                               //save last requested ROI coordinates
                               //-----------------------------------
                               #center_x_old        :=  #set_center_x;
                               #center_y_old        :=  #set_center_y;
                               #outer_radius_old    :=  #set_outer_radius;
                               #inner_radius_old    :=  #set_inner_radius;
                               #start_angle_old     :=  #set_start_angle;
                               #stop_angle_old      :=  #set_stop_angle;
                            END_IF;
                       END_IF;

                   //stero camera mode
                   //-----------------
                   ELSE
                       //ROI stereo camera 1
                       //-------------------
                       #set_ctr_x_scam_1    :=  "CM_INSELECT"(auto    :=  "APC".AUTOMATIC,              // area in x-dimension
                                                           track   :=  TRUE,
                                                           ac      :=  ROUND("AC".SET_ROI_CTR_X_SCAM),
                                                           kya     :=  "KYA".SET_ROI_CTR_X_SCAM);

                       #set_ctr_y_scam_1    :=  "CM_INSELECT"(auto    :=  "APC".AUTOMATIC,              //area in y-dimension
                                                           track   :=  TRUE,
                                                           ac      :=  ROUND("AC".SET_ROI_CTR_Y_SCAM),
                                                           kya     :=  "KYA".SET_ROI_CTR_Y_SCAM);

                       #set_width_scam_1    :=  "CM_INSELECT"(auto    :=  "APC".AUTOMATIC,              //sensor width
                                                           track   :=  TRUE,
                                                           ac      :=  ROUND("AC".SET_SEN_HGT),      //sensor rotated 90? height and width exchanged
                                                           kya     :=  "KYA".SET_ROI_HGT_SCAM);

                       #set_height_scam_1   :=  "CM_INSELECT"(auto    :=  "APC".AUTOMATIC,              //sensor height
                                                           track   :=  TRUE,
                                                           ac      :=  ROUND("AC".SET_SEN_WDH),      //sensor rotated 90? height and width exchanged
                                                           kya     :=  "KYA".SET_ROI_WDH_SCAM);

                       //check if ROI coordinate change is requested
                       //-------------------------------------------
                       IF NOT #O_NEW_ROI_CRD  THEN
                           //sensor position change stereo camera 1
                           //--------------------------------------
                           IF  (#set_ctr_x_scam_1 <> #set_ctr_x_scam_1_old)  OR
                               (#set_ctr_y_scam_1 <> #set_ctr_y_scam_1_old)  OR
                               (#set_width_scam_1 <> #set_width_scam_1_old)  OR
                               (#set_height_scam_1 <> #set_height_scam_1_old)    THEN 

                               #new_roi_crd :=  true;

                               //convert parameter values in string variables
                               //-------------------------------------------- 
                               #ctr_x_scam1     :=  DINT_TO_STRING (IN:= REAL_TO_DINT(#set_ctr_x_scam_1 * 100));
                               #ctr_y_scam1     :=  DINT_TO_STRING (IN:= REAL_TO_DINT(#set_ctr_y_scam_1 * 100));    
                               #width_scam1     :=  DINT_TO_STRING (IN:= REAL_TO_DINT(#set_width_scam_1 * 100));
                               #height_scam1    :=  DINT_TO_STRING (IN:= REAL_TO_DINT(#set_height_scam_1 * 100));    

                           END_IF;
                           //evaluate new ROI coordinate command string
                           //------------------------------------------
                           IF #new_roi_crd THEN

                               //delete ROI coordinate string
                               //----------------------------   
                               #roi_crd_strg := DELETE(IN:= #roi_crd_strg, L:= 60, P:= 0);

                               //built new ROI coordinate string
                               //-------------------------------     
                               #roi_crd_strg    := CONCAT(IN1:= 'rke1_cc=' , IN2:= #ctr_x_scam1);

                               #roi_crd_strg    := CONCAT(IN1:= #roi_crd_strg, IN2:= #delimiter);

                               #roi_crd_strg    := CONCAT(IN1:= #roi_crd_strg, IN2:= #ctr_y_scam1);

                               #roi_crd_strg    := CONCAT(IN1:= #roi_crd_strg, IN2:= #delimiter);

                               #roi_crd_strg    := CONCAT(IN1:= #roi_crd_strg, IN2:= #width_scam1);

                               #roi_crd_strg    := CONCAT(IN1:= #roi_crd_strg, IN2:= #delimiter);

                               #roi_crd_strg    := CONCAT(IN1:= #roi_crd_strg, IN2:= #height_scam1);

                               #O_ROI_CRD_STRG  :=  #roi_crd_strg;    //write new ROI coordinate string
                               #O_NEW_ROI_CRD   :=  true;

                               //save last requested ROI coordinates
                               //-----------------------------------
                               #set_ctr_x_scam_1_old    :=  #set_ctr_x_scam_1;
                               #set_ctr_y_scam_1_old    :=  #set_ctr_y_scam_1;
                               #set_width_scam_1_old    :=  #set_width_scam_1;
                               #set_height_scam_1_old   :=  #set_height_scam_1;
                           END_IF;
                       END_IF;

                       //ROI stereo camera 2
                       //-------------------
                       #set_ctr_x_scam_2    :=  #set_ctr_x_scam_1 + "PAR_SUB".CTR_X_SCAM_2_ADJ;
                       #set_ctr_y_scam_2    :=  #set_ctr_y_scam_1 + "PAR_SUB".CTR_Y_SCAM_2_ADJ;
                       #set_width_scam_2    :=  #set_width_scam_1;
                       #set_height_scam_2   :=  #set_height_scam_1;

                       //check if ROI coordinate change is requested
                       //-------------------------------------------
                       IF NOT #O_NEW_ROI_CRD  THEN
                           //sensor position change stereo camera 2
                           //--------------------------------------
                           IF  (#set_ctr_x_scam_2 <> #set_ctr_x_scam_2_old)  OR
                               (#set_ctr_y_scam_2 <> #set_ctr_y_scam_2_old)  OR
                               (#set_width_scam_2 <> #set_width_scam_2_old)  OR
                               (#set_height_scam_2 <> #set_height_scam_2_old)    THEN 

                               #new_roi_crd :=  true;

                               //convert parameter values in string variables
                               //-------------------------------------------- 
                               #ctr_x_scam2     :=  DINT_TO_STRING (IN:= REAL_TO_DINT(#set_ctr_x_scam_2 * 100));
                               #ctr_y_scam2     :=  DINT_TO_STRING (IN:= REAL_TO_DINT(#set_ctr_y_scam_2 * 100));    
                               #width_scam2     :=  DINT_TO_STRING (IN:= REAL_TO_DINT(#set_width_scam_2 * 100));
                               #height_scam2    :=  DINT_TO_STRING (IN:= REAL_TO_DINT(#set_height_scam_2 * 100));    

                           END_IF;
                           //evaluate new ROI coordinate command string
                           //------------------------------------------
                           IF #new_roi_crd THEN

                               //delete ROI coordinate string
                               //----------------------------   
                               #roi_crd_strg := DELETE(IN:= #roi_crd_strg, L:= 60, P:= 0);

                               //built new ROI coordinate string
                               //-------------------------------     
                               #roi_crd_strg    := CONCAT(IN1:= 'rke2_cc=' , IN2:= #ctr_x_scam2);

                               #roi_crd_strg    := CONCAT(IN1:= #roi_crd_strg, IN2:= #delimiter);

                               #roi_crd_strg    := CONCAT(IN1:= #roi_crd_strg, IN2:= #ctr_y_scam2);

                               #roi_crd_strg    := CONCAT(IN1:= #roi_crd_strg, IN2:= #delimiter);

                               #roi_crd_strg    := CONCAT(IN1:= #roi_crd_strg, IN2:= #width_scam2);

                               #roi_crd_strg    := CONCAT(IN1:= #roi_crd_strg, IN2:= #delimiter);

                               #roi_crd_strg    := CONCAT(IN1:= #roi_crd_strg, IN2:= #height_scam2);

                               #O_ROI_CRD_STRG  :=  #roi_crd_strg;    //write new ROI coordinate string
                               #O_NEW_ROI_CRD   :=  true;

                               //save last requested ROI coordinates
                               //-----------------------------------
                               #set_ctr_x_scam_2_old    :=  #set_ctr_x_scam_2;
                               #set_ctr_y_scam_2_old    :=  #set_ctr_y_scam_2;
                               #set_width_scam_2_old    :=  #set_width_scam_2;
                               #set_height_scam_2_old   :=  #set_height_scam_2;
                           END_IF;
                       END_IF;
                   END_IF;        

               //rectangle ROI is selected
               //-------------------------
               ELSIF "LT".CAM_PRD_1_SEL THEN
                   #set_center_x    :=  "CM_INSELECT"(auto    :=  "APC".AUTOMATIC,              // area in x-dimension
                                                   track   :=  TRUE,
                                                   ac      :=  ROUND("AC".SET_SEN_CTR_X),
                                                   kya     :=  "KYA".SET_SEN_CTR_X_P1);

                   #set_center_y    :=  "CM_INSELECT"(auto    :=  "APC".AUTOMATIC,              //area in y-dimension
                                                   track   :=  TRUE,
                                                   ac      :=  ROUND("AC".SET_SEN_CTR_Y),
                                                   kya     :=  "KYA".SET_SEN_CTR_Y_P1);

                   #set_width       :=  "CM_INSELECT"(auto    :=  "APC".AUTOMATIC,              //sensor width
                                                   track   :=  TRUE,
                                                   ac      :=  ROUND("AC".SET_SEN_WDH),
                                                   kya     :=  "KYA".SET_SEN_WDH_P1);


                   #set_height       :=  "CM_INSELECT"(auto   :=  "APC".AUTOMATIC,              //sensor height
                                                   track   :=  TRUE,
                                                   ac      :=  ROUND("AC".SET_SEN_HGT),
                                                   kya     :=  "KYA".SET_SEN_HGT_P1);


                   //check if ROI coordinate change is requested
                   //-------------------------------------------
                   IF NOT #O_NEW_ROI_CRD  THEN
                       //melting detection
                       //-----------------
                       IF  (#set_center_x <> #center_x_old)  OR
                           (#set_center_y <> #center_y_old)  OR
                           (#set_width <> #width_old)        OR
                           (#set_height <> #height_old)      THEN 

                           #new_roi_crd :=  true;

                           //convert parameter values in string variables
                           //-------------------------------------------- 
                           #center_x    :=  DINT_TO_STRING (IN:= REAL_TO_DINT(#set_center_x * 100));
                           #center_y    :=  DINT_TO_STRING (IN:= REAL_TO_DINT(#set_center_y * 100));    
                           #width       :=  DINT_TO_STRING (IN:= REAL_TO_DINT(#set_width * 100));
                           #height      :=  DINT_TO_STRING (IN:= REAL_TO_DINT(#set_height * 100));    

                       END_IF;
                   END_IF;

                   //evaluate new ROI coordinate command string
                   //------------------------------------------
                   IF #new_roi_crd THEN

                       //delete ROI coordinate string
                       //----------------------------   
                       #roi_crd_strg := DELETE(IN:= #roi_crd_strg, L:= 60, P:= 0);

                       //built new ROI coordinate string
                       //-------------------------------     
                       #roi_crd_strg    := CONCAT(IN1:= 'rec_crd=' , IN2:= #center_x);

                       #roi_crd_strg    := CONCAT(IN1:= #roi_crd_strg, IN2:= #delimiter);

                       #roi_crd_strg    := CONCAT(IN1:= #roi_crd_strg, IN2:= #center_y);

                       #roi_crd_strg    := CONCAT(IN1:= #roi_crd_strg, IN2:= #delimiter);

                       #roi_crd_strg    := CONCAT(IN1:= #roi_crd_strg, IN2:= #width);

                       #roi_crd_strg    := CONCAT(IN1:= #roi_crd_strg, IN2:= #delimiter);

                       #roi_crd_strg    := CONCAT(IN1:= #roi_crd_strg, IN2:= #height);

                       #O_ROI_CRD_STRG  :=  #roi_crd_strg;    //write new ROI coordinate string
                       #O_NEW_ROI_CRD   :=  true;

                       //save last requested ROI coordinates
                       //-----------------------------------
                       #center_x_old    :=  #set_center_x;
                       #center_y_old    :=  #set_center_y;
                       #width_old       :=  #set_width;
                       #height_old      :=  #set_height;

                   END_IF;
               END_IF; 
           END_IF;

           //reset flag new ROI coordinates
           //------------------------------
           #new_roi_crd :=  false;

           //melt vibration measurement - acitve in all measurement methods
           //--------------------------------------------------------------
           //read settings of melt vibration sensor from recipe or manual input 
           //------------------------------------------------------------------
           #set_mlt_vib_center_x    :=  "KYA".SET_SEN_MLT_VIB_CTR_X;          //area in y-dimension

           #set_mlt_vib_center_y    :=  "KYA".SET_SEN_MLT_VIB_CTR_Y;          //area in y-dimension

           #set_mlt_vib_width       :=  "KYA".SET_SEN_MLT_VIB_WDH;            //senor width

           //check if ROI coordinate change is requested
           //-------------------------------------------
           IF NOT #O_NEW_ROI_CRD  THEN
               //melt vibration measurement
               //--------------------------
               IF (#set_mlt_vib_center_x <> #mlt_vib_center_x_old)  OR
                  (#set_mlt_vib_center_y <> #mlt_vib_center_y_old)  OR
                  (#set_mlt_vib_width <> #mlt_vib_width_old)        THEN 

                   #new_mlt_vib_roi_crd :=  true;

                   //convert parameter values in string variables
                   //-------------------------------------------- 
                   #mlt_vib_center_x    :=  DINT_TO_STRING (IN:= REAL_TO_DINT(#set_mlt_vib_center_x * 100));
                   #mlt_vib_center_y    :=  DINT_TO_STRING (IN:= REAL_TO_DINT(#set_mlt_vib_center_y * 100));    
                   #mlt_vib_width       :=  DINT_TO_STRING (IN:= REAL_TO_DINT(#set_mlt_vib_width * 100));

               END_IF; 
           END_IF;       

           //evaluate new melt vibration ROI coordinate command string
           //---------------------------------------------------------
           IF #new_mlt_vib_roi_crd THEN

               //delete ROI coordinate string
               //----------------------------   
               #roi_crd_strg := DELETE(IN:= #roi_crd_strg, L:= 60, P:= 0);

               //built new ROI coordinate string
               //-------------------------------     
               #roi_crd_strg    := CONCAT(IN1:= 'vib_crd=' , IN2:= #mlt_vib_center_x);

               #roi_crd_strg    := CONCAT(IN1:= #roi_crd_strg, IN2:= #delimiter);

               #roi_crd_strg    := CONCAT(IN1:= #roi_crd_strg, IN2:= #mlt_vib_center_y);

               #roi_crd_strg    := CONCAT(IN1:= #roi_crd_strg, IN2:= #delimiter);

               #roi_crd_strg    := CONCAT(IN1:= #roi_crd_strg, IN2:= #mlt_vib_width);

               #O_ROI_CRD_STRG  :=  #roi_crd_strg;    //write new ROI coordinate string
               #O_NEW_ROI_CRD   :=  true;

               //save last requested ROI coordinates
               //-----------------------------------
               #mlt_vib_center_x_old    :=  #set_mlt_vib_center_x;
               #mlt_vib_center_y_old    :=  #set_mlt_vib_center_y;
               #mlt_vib_width_old       :=  #set_mlt_vib_width;

               //reset flag new melt vibration ROI coordinates
               //---------------------------------------------
               #new_mlt_vib_roi_crd :=  false;

           END_IF;     

           //evaluate recipe threshold setpoint
           //----------------------------------
           #ac_set_sen_thr  :=  ROUND("AC".SET_SEN_THR * 10.0);   //shift decimal place one digit to the right and round

           #ac_set_sen_thr  :=  #ac_set_sen_thr / 10.0;          //shift decimal place one digit to the left 

           //evaluate recipe threshold setpoint for camera 2
           //----------------------------------
           #ac_set_sen_thr_2  :=  ROUND("AC".SET_CAM_2_THR * 10.0);   //shift decimal place one digit to the right and round

           #ac_set_sen_thr_2  :=  #ac_set_sen_thr_2 / 10.0;          //shift decimal place one digit to the left 

           //evaluate threshold setpoint mode related
           //----------------------------------------
           IF "LT".CAM_MLT   THEN
               //read sensor threshold
               //---------------------
               #set_thr :=  "CM_INSELECT"(auto    :=  "APC".AUTOMATIC,              
                                       track   :=  TRUE,
                                       ac      :=  #ac_set_sen_thr,             //use rounded value
                                       kya     :=  "KYA".SET_SEN_THR_P4);

               //set command identifier
               //----------------------
               #thr_cmd         :=  'mlt_thr=';

           ELSIF "LT".CAM_DIP   THEN
               //read sensor threshold
               //---------------------
               #set_thr :=  "CM_INSELECT"(auto    :=  "APC".AUTOMATIC,              
                                       track   :=  TRUE,
                                       ac      :=  #ac_set_sen_thr,             //use rounded value
                                       kya     :=  "KYA".SET_SEN_THR_P3);

               //set command identifier
               //----------------------
               #thr_cmd         :=  'dip_thr=';

           ELSIF "LT".CAM_DIA   THEN
               //read threshold of seqmented circle ROI
               //--------------------------------------           
               IF "LT".CAM_PRD_2_SEL THEN 
                   //threshold
                   //---------
                   #set_thr :=  "CM_INSELECT"(auto    :=  "APC".AUTOMATIC,              
                                           track   :=  TRUE,
                                           ac      :=  #ac_set_sen_thr,             //use rounded value
                                           kya     :=  "KYA".SET_SEN_THR_P2);

                   //set circle sensor command identifier
                   //------------------------------------
                   #thr_cmd         :=  'dia_thr=';

                   //stereo camera installed
                   //-----------------------
                   IF (("CNF".ACT_DVC_CNF AND 2#0000_0000_0000_1000_0000_0000_0000_0000) = 2#0000_0000_0000_1000_0000_0000_0000_0000) THEN  
                       //shoulder phase
                       //--------------
                       IF ("APC".STATUS = "APC".SHOULDER) THEN
                           //threshold - used for a second camera only in shoulder phase
                           //-----------------------------------------------------------
                           #set_thr_2 :=  "CM_INSELECT"(auto    :=  "APC".AUTOMATIC,              
                                                     track   :=  TRUE,
                                                     ac      :=  #ac_set_sen_thr_2,             //use rounded value
                                                     kya     :=  "KYA".SET_CAM_2_THR);

                           //set circle sensor command identifier
                           //------------------------------------
                           #thr_cmd_2        :=  'diathr2=';
                       //other phases
                       //------------
                       ELSE
                           "KYA".SET_CAM_2_THR   := #set_thr; //track KYA value of second threshold with first threshold      
                       END_IF;
                   END_IF;    
               //read threshold of rectangle ROI
               //-------------------------------
               ELSIF "LT".CAM_PRD_1_SEL  THEN 
                   #set_thr :=  "CM_INSELECT"(auto    :=  "APC".AUTOMATIC,              
                                           track   :=  TRUE,
                                           ac      :=  #ac_set_sen_thr,             //use rounded value
                                           kya     :=  "KYA".SET_SEN_THR_P1);

                   //set circle sensor command identifier
                   //------------------------------------
                   #thr_cmd         :=  'rec_thr=';

               END_IF;
           END_IF;

           //read melt vibration sensor threshold
           //------------------------------------
           #set_mlt_vib_thr :=  "KYA".SET_SEN_MLT_VIB_THR;

           //check if ROI threshold change is requested
           //------------------------------------------
           IF NOT #O_NEW_ROI_THR THEN
               //melting, dipping or diameter measurement
               //----------------------------------------
               IF (#set_thr <> #thr_old) THEN 
                   #new_thr_req :=  true;

                   //convert parameter values in string variables
                   //-------------------------------------------- 
                   #thr :=  INT_TO_STRING (IN:= REAL_TO_INT(#set_thr * 100));      //circle sensor, dip line or junk detection

               //melt vibration measurement
               //--------------------------
               ELSIF (#set_mlt_vib_thr <> #mlt_vib_thr_old) THEN
                   #new_mlt_vib_thr_req :=  true;

                   //convert melt vibration threshold parameter value in string variable
                   //------------------------------------------------------------------- 
                   #mlt_vib_thr :=  INT_TO_STRING (IN:= REAL_TO_INT(#set_mlt_vib_thr * 100));

               END_IF; 
           END_IF;

           //check if ROI threshold change is requested for camera 2
           //------------------------------------------
           IF NOT #O_NEW_ROI_THR_2 THEN
               //melting, dipping or diameter measurement
               //----------------------------------------

               IF (#set_thr_2 <> #thr_old_2) THEN 
                   #new_thr_req_2 :=  true;

                   //convert parameter values in string variables
                   //-------------------------------------------- 
                   #thr_2 :=  INT_TO_STRING (IN:= REAL_TO_INT(#set_thr_2 * 100));      //circle sensor, dip line or junk detection

               END_IF;        
           END_IF;

           //evaluate new ROI threshold command string
           //-----------------------------------------
           IF #new_thr_req THEN                         //melting, dipping or diameter measurement

               //delete command string
               //---------------------   
               #roi_thr_strg := DELETE(IN:= #roi_thr_strg, L:= 20, P:= 0);

               //built new command string
               //------------------------     
               #roi_thr_strg    := CONCAT(IN1:= #thr_cmd, IN2:= #thr);

               #O_ROI_THR_STRG  :=  #roi_thr_strg;    //write new ROI threshold string
               #O_NEW_ROI_THR   :=  true;

               //save last requested sensor threshold parameter
               //----------------------------------------------
               #thr_old :=  #set_thr;

               //reset new sensor shape flag
               //--------------------------- 
               #new_thr_req :=  false;


           ELSIF #new_mlt_vib_thr_req THEN              //melt vibration measurement

               //delete command string
               //---------------------   
               #roi_thr_strg := DELETE(IN:= #roi_thr_strg, L:= 20, P:= 0);

               //built new command string
               //------------------------     
               #roi_thr_strg    := CONCAT(IN1:= 'vib_thr=', IN2:= #mlt_vib_thr);

               #O_ROI_THR_STRG  :=  #roi_thr_strg;    //write new ROI threshold string
               #O_NEW_ROI_THR   :=  true;

               //save last requested sensor threshold parameter
               //----------------------------------------------
               #mlt_vib_thr_old :=  #set_mlt_vib_thr;

               //reset new sensor shape flag
               //--------------------------- 
               #new_mlt_vib_thr_req :=  false;


           END_IF;

           //evaluate new ROI threshold command string for camnera 2
           //-----------------------------------------

           IF #new_thr_req_2 THEN                         //melting, dipping or diameter measurement

               //delete command string
               //---------------------   
               #roi_thr_strg_2 := DELETE(IN:= #roi_thr_strg_2, L:= 20, P:= 0);

               //built new command string
               //------------------------     
               #roi_thr_strg_2    := CONCAT(IN1:= #thr_cmd_2, IN2:= #thr_2);

               #O_ROI_THR_STRG_2  :=  #roi_thr_strg_2;    //write new ROI threshold string
               #O_NEW_ROI_THR_2   :=  true;

               //save last requested sensor threshold parameter
               //----------------------------------------------
               #thr_old_2 :=  #set_thr_2;

               //reset new sensor shape flag
               //--------------------------- 
               #new_thr_req_2 :=  false;
           END_IF;


       END_IF;
END_FUNCTION_BLOCK

FUNCTION_BLOCK "CHAR_TO_DINT"   // FB104, SCL
{ S7_Optimized_Access := 'FALSE' }
VERSION : 0.0
// --------------------------------------------------------------------------------
//     program     :    CHAR_TO_DINT
//     description :    convert characters to double integer      
//     name        :    G. Eibelsh鋟ser
//     date        :    11.05.2010
// 
//     revision    :
//     name        :
//     date        :    
//                     (c)PVA Tepla AG
//     --------------------------------------------------------------------------------
   VAR_INPUT
      I_AMT_OF_BYTES : Int;
   END_VAR
   VAR_OUTPUT
      O_CAM_VALUE : Array[0..19] of DInt;   // increased for stereo camera test
   END_VAR
   VAR
      i : Int;
      k : Int;
      digit : Int;
      number : DInt;
   END_VAR
BEGIN

       //init temporary function variables
       //---------------------------------
       #digit      := 0;                                   
       #number     := 0;
       #k          := 0;

       FOR #i:= 4 TO (#I_AMT_OF_BYTES) DO        //exclude first four characters in data DB                             
           //last character detected - abort calculation and function
           //--------------------------------------------------------
           IF "BM_CAM_EVAL_DB".Data[#i] = BYTE_TO_CHAR(B#16#D) THEN        //exit conversion when carriage return appears in telegram
               #O_CAM_VALUE[#k] := #number;
               EXIT;
           ELSE
               //delimter detected - abort calculation of value
               //----------------------------------------------
               IF ("BM_CAM_EVAL_DB".Data[#i] = ';')THEN             
                   #O_CAM_VALUE[#k]  := #number;
                   #k               := #k + 1;                               //increase value counter
                   #number          := 0;
                   #digit           := 0;
               //calculate double integer from characters byte wise
               //--------------------------------------------------
               ELSE
                   #digit := CHAR_TO_INT("BM_CAM_EVAL_DB".Data[#i])-48;   // convert ASCII character in integer value
                   #number   := #number * 10 + #digit;                       
               END_IF;
           END_IF;
       END_FOR;
END_FUNCTION_BLOCK

FUNCTION_BLOCK "BM_MOB_FDR_MAIN"   // FB105, SCL
{ S7_Optimized_Access := 'FALSE' }
VERSION : 0.0
// --------------------------------------------------------------------------------
//     program     :   BM_MOB_FDR_MAIN
//     description :   main control of mobile feeder
//     name        :   G. Eibelsh鋟ser
//     date        :   26.10.2011
//   
//     revision    :
//     name        :
//     date        :    
//                     (c)PVATePla AG
//     --------------------------------------------------------------------------------
   VAR
      i : Int;
   END_VAR
   VAR_TEMP
      dbl_srv_mode : Bool;
   END_VAR
BEGIN

       //ReadStatus from feeder
       //-------------------------------------------------------------------------
       "DV".CB_FLT_AC230V_FDR  := DWORD_TO_DINT("P_BM_FDR_STAT":P AND 2#0000_0000_0000_0001)<>0;
       "DV".CB_FLT_DC24V_FDR   := DWORD_TO_DINT("P_BM_FDR_STAT":P AND 2#0000_0000_0000_0010)<>0;
       "DV".FDR_CH_HOME_POS    := DWORD_TO_DINT("P_BM_FDR_STAT":P AND 2#0000_0000_0000_0100)<>0;
       "DV".FDR_CH_FDG_POS     := DWORD_TO_DINT("P_BM_FDR_STAT":P AND 2#0000_0000_0000_1000)<>0;
       "DV".FDR_TUBE_HOME_POS  := DWORD_TO_DINT("P_BM_FDR_STAT":P AND 2#0000_0000_0001_0000)<>0;
       "DV".FDR_TUBE_FCH_POS   := DWORD_TO_DINT("P_BM_FDR_STAT":P AND 2#0000_0000_0010_0000)<>0;
       "DV".FDR_TUBE_FDG_POS   := DWORD_TO_DINT("P_BM_FDR_STAT":P AND 2#0000_0000_0100_0000)<>0;
       "DV".FDR_IN_POS         := DWORD_TO_DINT("P_BM_FDR_STAT":P AND 2#0000_0000_1000_0000)<>0;

       //                      := DV.FDR_VIB_ENB  

       //reset feeder undocking done flag when feeder is electrically disconnected
       //-------------------------------------------------------------------------
       IF NOT "DV".MOB_FDR_CON    THEN 
           "LT".MOB_FDR_UDCK_DONE    :=  FALSE; 
           "DV".MOB_FDR_PB_TRM       :=  FALSE;               
           #i                       :=  0;

       //reset mobile feeder connection flag before electrical disconnection
       //-------------------------------------------------------------------
       ELSIF "LT".MOB_FDR_UDCK_DONE THEN
           //IF BYTE_TO_INT(PEB256)<>0 THEN
           //    DV.MOB_FDR_PB_TRM   :=  FALSE;
           //END_IF;                  
           #i   :=  0;

       //set mobile feeder connection flag
       //---------------------------------
       ELSIF "DV".MOB_FDR_CON THEN                  //electrical connection done
           IF (#i > 50) THEN 
               "DV".MOB_FDR_PB_TRM   :=  TRUE;       //termination flag 5s delayed               
           ELSE
               IF "SysTick100ms" THEN 
                   #i   :=  #i + 1;
               END_IF;
           END_IF;
       END_IF;

       //electrical connection of mobile feeder done
       //-------------------------------------------
       "LT".MOB_FDR_EL_CON_DONE  :=  "DV".MOB_FDR_PB_TRM;

       //disable service mode when sequences are active
       //----------------------------------------------
       #dbl_srv_mode    :=  "APC".AUTOMATIC OR "LT".MOB_FDR_DCK_ATV OR "LT".MOB_FDR_UDCK_ATV OR "LT".MOB_FDR_MVE_IN_SEQ_ON OR "LT".MOB_FDR_MVE_OUT_SEQ_ON;

       //activate/deactivate service mode of mobile feeder
       //-------------------------------------------------
       IF #dbl_srv_mode THEN 
           "LT".MOB_FDR_SRV_ON :=    FALSE;
       ELSE
           "LT".MOB_FDR_SRV_ON := ("KYD".MOB_FDR_SRV_ON OR "LT".MOB_FDR_SRV_ON) AND NOT "KYD".MOB_FDR_SRV_OFF;
       END_IF;

       //call mobile feeder modules
       //--------------------------
       IF "DV".MOB_FDR_CALL THEN 
           //service function activated
           //--------------------------
           IF "LT".MOB_FDR_SRV_ON THEN
               //call mobile feeder service function
               //-----------------------------------
               "BM_MOB_FDR_SRV"();
           ELSE            
               //call mobile feeder drive sequence function block
               //------------------------------------------------
               "BM_MOB_FDR_DRV_SEQ_DB"();

           END_IF; 

           //set circuit breaker alarm messages of mobile feeder
           //---------------------------------------------------
           "FLT".MOB_FDR_CB_AC_230V  := "DV".CB_FLT_AC230V_FDR;

           "FLT".MOB_FDR_CB_DC_24V   := "DV".CB_FLT_DC24V_FDR;                

           //write status variables
           //----------------------
           "LT".MOB_FDR_CH_HOME_POS  :=  "DV".FDR_CH_HOME_POS;
           "LT".MOB_FDR_TUBE_HOME_POS:=  "DV".FDR_TUBE_HOME_POS;
           "LT".MOB_FDR_TUBE_FCH_POS :=  "DV".FDR_TUBE_FCH_POS;
           "LT".MOB_FDR_CH_FDG_POS   :=  "DV".FDR_CH_FDG_POS;
           "LT".MOB_FDR_TUBE_FDG_POS :=  "DV".FDR_TUBE_FDG_POS;
           "LT".FDR_LS_TUBE_OUT      :=  "DV".FDR_TUBE_HOME_POS;    //used for tube symbol in EKZ Explorer

           //write display values of mobile feeder
           //-------------------------------------
           "DIS".MOB_FDR_ACT_TUBE_TMP    :=  0.0;
           "DIS".MOB_FDR_ACT_TUBE_POS    :=  "P_BM_FDR_ACT_TUBE_POS":P;
           "DIS".ACT_LEAKR_FDR           :=  "AV".MOB_FDR_LKR;    //AV.AVG_FDG_RTE; 
           "DIS".ACT_PRS_DROP_FDR        :=  "AV".ACT_PRS_DROP_FDR;
           "DIS".MOB_FDR_ACT_CRG_LVL     :=  "P_BM_FDR_ACT_CRG_LVL":P;

       ELSE
           //reset circuit breaker alarm messages of mobile feeder
           //---------------------------------------------------
           "FLT".MOB_FDR_CB_AC_230V      :=  FALSE;
           "FLT".MOB_FDR_CB_DC_24V       :=  FALSE;

           "FLT".MOB_FDR_INIT_KL_3312    :=  FALSE;  
           "FLT".MOB_FDR_TC_TUBE         :=  FALSE;  
           "FLT".MOB_FDR_INIT_KL2552     :=  FALSE; 
           "FLT".MOB_FDR_MOV_IN_SEQ_ABR  :=  FALSE; 
           "FLT".MOB_FDR_MOV_OUT_SEQ_ABR :=  FALSE; 
           "FLT".MOB_FDR_DCK_SEQ_ABR     :=  FALSE;
           "FLT".MOB_FDR_UDCK_SEQ_ABR    :=  FALSE;
           "FLT".MOB_FDR_FNC_PRS_HI      :=  FALSE;
           "FLT".MOB_FDR_PRS_HI          :=  FALSE;
           "FLT".FEED_RTE_TOO_HI         :=  FALSE;

           //reset vacuum control flags
           //--------------------------
           "DV".MOB_FDR_P3_ON_REQ        :=  FALSE;
           "DV".MOB_FDR_V3_2_OPN_REQ     :=  FALSE;
           "DV".MOB_FDR_V24_OPN_REQ      :=  FALSE;

           //reset status variables
           //----------------------
           "LT".MOB_FDR_CH_HOME_POS  :=  FALSE;
           "LT".MOB_FDR_TUBE_HOME_POS:=  FALSE;

           "LT".MOB_FDR_TUBE_FCH_POS :=  FALSE;

           "LT".MOB_FDR_CH_FDG_POS   :=  FALSE;
           "LT".MOB_FDR_TUBE_FDG_POS :=  FALSE;

           "LT".MOB_FDR_TUBE_DN      :=  FALSE;
           "LT".MOB_FDR_TUBE_UP      :=  FALSE;
           "LT".MOB_FDR_TUBE_STOP    :=  FALSE;
           "LT".MOB_FDR_CH_SW_R      :=  FALSE;
           "LT".MOB_FDR_CH_SW_L      :=  FALSE;
           "LT".MOB_FDR_CH_SW_STOP   :=  FALSE;

           //reset display values of mobile feeder
           //-------------------------------------
           "DIS".MOB_FDR_ACT_TUBE_POS    :=  0.0;
           "DIS".MOB_FDR_SET_VIB_FRQ     :=  0.0;
           "DIS".MOB_FDR_ACT_CRG_LVL     :=  0.0;
           "DIS".ACT_STD_DEV_FILL_LVL    :=  0.0;

           //call mobile feeder service function
           //-----------------------------------
           IF "LT".MOB_FDR_SRV_ON THEN
               "BM_MOB_FDR_SRV"();
           END_IF;
       END_IF;


       //check if mobile feeder is located on puller flange
       //--------------------------------------------------
       IF "DV".FDR_IN_POS THEN
           IF NOT "LT".MOB_FDR_IN_POS THEN 
               //reset mobile feeder docking and drive sequence variables
               //-------------------------------------------------------- 
               "LT".MOB_FDR_DCK_ATV          :=  FALSE;
               "LT".MOB_FDR_UDCK_ATV         :=  FALSE;
               "LT".MOB_FDR_DCK_DONE         :=  FALSE;
               "LT".MOB_FDR_UDCK_DONE        :=  FALSE;
               "LT".MOB_FDR_MVE_OUT_SEQ_ON   :=  FALSE;
               "LT".MOB_FDR_MVE_IN_SEQ_ON    :=  FALSE;
               "LT".MOB_FDR_MVE_SEQ_ARB      :=  FALSE;        
               "LT".MOB_FDR_TUBE_DN          :=  FALSE;
               "LT".MOB_FDR_TUBE_UP          :=  FALSE;
               "LT".MOB_FDR_TUBE_STOP        :=  FALSE;
               "LT".MOB_FDR_CH_SW_R          :=  FALSE;
               "LT".MOB_FDR_CH_SW_L          :=  FALSE;
               "LT".MOB_FDR_CH_SW_STOP       :=  FALSE;
               "LT".MOB_FDR_VIB_ON           :=  FALSE;
           END_IF;
           "LT".MOB_FDR_IN_POS   :=  TRUE;
       ELSE
           "LT".MOB_FDR_IN_POS   :=  FALSE;
       END_IF;
END_FUNCTION_BLOCK

FUNCTION_BLOCK "BM_MOB_FDR_DCK"   // FB106, SCL
{ S7_Optimized_Access := 'FALSE' }
VERSION : 0.0
// --------------------------------------------------------------------------------
//     program     :   BM_MOB_FDR_DCK
//     description :   docking of mobile feeder to puller
//     name        :   G. Eibelsh鋟ser
//     date        :   26.10.2011
//   
//     revision    :
//     name        :
//     date        :    
//                     (c)PVATePla AG
//     --------------------------------------------------------------------------------
   VAR
      arb_dck_seq : Bool;
      "step" : Int;
      i : Int;
      j : Int;
      prg_cnt : Int;
      mob_fdr_prs_bfe_lt : Real;
   END_VAR
BEGIN

       //set mobile feeder docking request 
       //---------------------------------
       IF          "LT".MOB_FDR_IN_POS                   //mobile feeder is in position
           AND NOT "LT".MOB_FDR_UDCK_ATV                 //undocking sequence is not running
           AND NOT "LT".MOB_FDR_DCK_DONE                 //docking sequence is not done
           AND NOT "LT".MOB_FDR_UDCK_DONE    THEN        //undocking sequence is not done - reseted after disconnection of plug

           IF "KYD".MOB_FDR_DCK_ON  THEN
               "LT".MOB_FDR_DCK_ATV  :=  TRUE;
           END_IF;
       END_IF;

       //abort mobile feeder docking sequence and vent feeder
       //----------------------------------------------------
       IF NOT "LT".MOB_FDR_DCK_DONE  AND NOT "FLT".MOB_FDR_DCK_SEQ_ABR THEN
           IF "LT".MOB_FDR_DCK_ATV AND "KYD".MOB_FDR_ARB_SEQ  THEN
               #arb_dck_seq  :=  true;
           END_IF;
       END_IF;

       //mobile feeder docking sequence
       //------------------------------
       IF "LT".MOB_FDR_DCK_ATV  THEN 

           //set step to abort docking sequence
           //----------------------------------
           IF (#arb_dck_seq AND (#step <> 90)) THEN
               #step    := 90;
           END_IF;

           //sequence steps
           //--------------
           CASE #step OF 

               0 : //initialisation step
                   //-------------------
                   #i                       :=  0;
                   #prg_cnt                 :=  0;
                   "AV".MOB_FDR_LKR          :=  0.0;
                   "AV".ACT_PRS_DROP_FDR     :=  0.0;
                   "FLT".ME_LEAK_TST_FDR     :=  FALSE;
                   "FLT".MOB_FDR_DCK_SEQ_ABR :=  FALSE;
                   "FLT".MOB_FDR_UDCK_SEQ_ABR:=  FALSE;
                   "FLT".MOB_FDR_PMP_TME     :=  FALSE;
                   "DV".MOB_FDR_V11_OPN_REQ  :=  FALSE;
                   "DV".MOB_FDR_V11_CLD_REQ  :=  TRUE;
                   "DV".FDG_MVE_IN_SEQ_DONE  :=  FALSE;
                   #step                    :=  #step + 10;

               10: //switch on vacuum pump P3 and open valve V3.2
                   //--------------------------------------------
                   "DV".MOB_FDR_P3_ON_REQ    :=  TRUE;
                   IF "SysTick1s"    THEN
                       #i := #i + 1;
                   END_IF;

                   IF (#i > 3) THEN                     //wait 
                       "DV".MOB_FDR_V3_2_OPN_REQ :=  TRUE;
                   END_IF;

                   IF ("DV".MOB_FDR_V3_2_OPN_REQ AND "PDO".V3_2) THEN                    //valve V3.2 opened
                       #step    :=  #step + 10;
                       #i       :=  0;
                       #j       :=  0;
                   END_IF;

               20: //pump down of mobile feeder
                   //--------------------------
                   IF (REAL_TO_INT("PAR_MAIN".MOB_FDR_DCK_PRG_CYC) > 0) THEN            //check amount of purge cycles 
                       IF ("AV".ACT_PRS_FDR <= "PAR_MAIN".MOB_FDR_DCK_PRG_PRS) THEN
                           #step    :=  #step + 10;
                       END_IF;
                       // Monitoring pump time
                       IF "SysTick1s" THEN
                          #j := #j+1;
                       END_IF;

                       IF (#j> REAL_TO_INT("PAR_MAIN".MOB_FDR_DCK_ALM_TME1)) THEN
                          "FLT".MOB_FDR_PMP_TME := ("AV".ACT_PRS_FDR > "PAR_MAIN".MOB_FDR_DCK_PRS_TRG1);
                       ELSE                  
                          "FLT".MOB_FDR_PMP_TME := False;
                       END_IF;
                       IF (#j> REAL_TO_INT("PAR_MAIN".MOB_FDR_DCK_ALM_TME2))THEN
                          "FLT".MOB_FDR_PMP_TME := ("AV".ACT_PRS_FDR > "PAR_MAIN".MOB_FDR_DCK_PRS_TRG2);
                       ELSE                  
                          "FLT".MOB_FDR_PMP_TME := False;
                       END_IF;

                   //pump down without purging
                   //-------------------------
                   ELSE
                       #step    :=  #step + 30;      //pump down to final pressure
                   END_IF;

               30: //close feeder vacuum valve V3.2
                   //------------------------------
                   "DV".MOB_FDR_V3_2_OPN_REQ :=  FALSE;
                   "FLT".MOB_FDR_PMP_TME := False;

                   IF "SysTick1s"    THEN
                       #i := #i + 1;
                   END_IF;

                   IF NOT "PDO".V3_2 THEN                    //valve V3.2 closed
                       IF (#i > 3) THEN                     //wait 
                           #step    :=  #step + 10;
                           #prg_cnt :=  #prg_cnt + 1;
                           #i       :=  0;
                       END_IF;
                   END_IF;

               40: //purge feeder
                   //------------       
                   IF (#i >= (REAL_TO_INT("PAR_MAIN".MOB_FDR_DCK_PRG_TME)) OR "DV".APS_FDR_DELAYED) THEN
                       "DV".MOB_FDR_V24_OPN_REQ :=  FALSE;
                   ELSE
                       "DV".MOB_FDR_V24_OPN_REQ :=  TRUE;
                   END_IF;

                   IF "SysTick1s"    THEN
                       #i := #i + 1;
                   END_IF;

                   IF NOT "DV".MOB_FDR_V24_OPN_REQ THEN 
                       IF NOT "PDO".V24 THEN
                           IF (#prg_cnt >= (REAL_TO_INT("PAR_MAIN".MOB_FDR_DCK_PRG_CYC))) THEN  
                               #step    :=  #step + 10;
                               #i       :=  0;
                           ELSE
                               #step    :=  #step - 30;     //repeat pump down and purging
                               #i       :=  0;
                           END_IF;
                       END_IF;     
                   END_IF;
                   #j  := 0;

               50: //pump down to final pressure
                   //---------------------------
                   IF ("AV".ACT_PRS_FDR <= "PAR_MAIN".MOB_FDR_DCK_FIN_PRS) THEN            //final pressure reached
                       IF "SysTick1s" THEN
                           #i := #i+1;
                       END_IF;
                       //wait time before leak test
                       //--------------------------
                       IF (#i >= (REAL_TO_INT("PAR_MAIN".MOB_FDR_DCK_WAIT_TME))) THEN
                           "DV".MOB_FDR_V3_2_OPN_REQ :=  FALSE;
                       END_IF;

                   ELSE
                       "DV".MOB_FDR_V3_2_OPN_REQ :=  TRUE;
                       #i                       :=  0;
                   END_IF;

                   IF NOT ("DV".MOB_FDR_V3_2_OPN_REQ OR "PDO".V3_2) THEN
                       #step    :=  #step + 10;
                       #i       :=  0;
                   END_IF;

                   // Monitoring pump time
                   IF "SysTick1s" THEN
                       #j := #j+1;
                   END_IF;

                   IF (#j> REAL_TO_INT("PAR_MAIN".MOB_FDR_DCK_ALM_TME1)) THEN
                       "FLT".MOB_FDR_PMP_TME := ("AV".ACT_PRS_FDR > "PAR_MAIN".MOB_FDR_DCK_PRS_TRG1);
                   ELSE                  
                       "FLT".MOB_FDR_PMP_TME := False;
                   END_IF;
                   IF (#j> REAL_TO_INT("PAR_MAIN".MOB_FDR_DCK_ALM_TME2))THEN
                       "FLT".MOB_FDR_PMP_TME := ("AV".ACT_PRS_FDR > "PAR_MAIN".MOB_FDR_DCK_PRS_TRG2);
                   ELSE                  
                       "FLT".MOB_FDR_PMP_TME := False;
                   END_IF;


               60: //wait 3 sec after vacuum valve V3.2 is closed and store actual pressure
                   //----------------------------------------------------------------------
                   #mob_fdr_prs_bfe_lt  := "AV".ACT_PRS_FDR; 
                   "FLT".MOB_FDR_PMP_TME := False;

                   IF "SysTick1s"    THEN
                       #i := #i + 1;
                   END_IF;

                   IF (#i > 3) THEN
                       "DV".MOB_FDR_P3_ON_REQ    :=  FALSE;          //switch off pump P3
                       #step                    :=  #step + 10;
                       #i                       :=  0;
                   END_IF;

               70: //leak test -> leakrate = (p2-p1)*V/t
                   //-----------------------------------
                   IF "SysTick1s"    THEN
                       #i := #i + 1;
                   END_IF;

                   //calculate leak rate
                   //-------------------
                   IF (#i > 0) THEN 
                       "AV".MOB_FDR_LKR := ("AV".ACT_PRS_FDR - #mob_fdr_prs_bfe_lt) * "CNF".VOLUME_MOB_FDR / (INT_TO_REAL(#i));
                   END_IF;

                   //keep leak rate on zero if calculation is negative
                   //-------------------------------------------------
                   IF ("AV".MOB_FDR_LKR < 0.0) THEN
                       "AV".MOB_FDR_LKR := 0.0;
                   END_IF;

                   //leak test time over
                   //-------------------
                   IF (#i >= (REAL_TO_INT("PAR_MAIN".MOB_FDR_DCK_LKT_TME))) THEN
                       #step    :=  #step + 10;
                   END_IF;

               80: //set alarm message if leak test failed
                   //-------------------------------------
                   IF ("AV".MOB_FDR_LKR > "PAR_MAIN".MOB_FDR_DCK_MAX_LKR) THEN
                       "FLT".ME_LEAK_TST_FDR :=  TRUE;

                       //repeat leak test
                       //----------------
                       IF "KYD".MOB_FDR_NEW_LKT   THEN
                           #step    :=  #step - 80;      //initialisation step 
                       END_IF;

                       //ignore bad leak rate
                       //--------------------
                       IF "KYD".MOB_FDR_IGN_LEAK_RTE   THEN
                           #step    :=  #step + 30;      //finish sequence
                       END_IF;

                       //abort sequence and vent feeder
                       //------------------------------
                       IF "KYD".MOB_FDR_ARB_SEQ   THEN
                           #step    :=  #step + 10;      //abort sequence
                       END_IF;

                   ELSE
                       #step    :=  #step + 30;          //finish sequence
                   END_IF;

               90: //abort docking sequence and vent feeder
                   //--------------------------------------
                   "DV".MOB_FDR_P3_ON_REQ    :=  FALSE;
                   "DV".MOB_FDR_V3_2_OPN_REQ :=  FALSE;
                   "FLT".MOB_FDR_DCK_SEQ_ABR :=  TRUE;
                   #arb_dck_seq             :=  false;

                   IF "DV".APS_FDR_DELAYED THEN                  //feeder at atmospheric pressure
                       "DV".MOB_FDR_V24_OPN_REQ  :=  FALSE;      //stop venting
                   ELSE 
                       "DV".MOB_FDR_V24_OPN_REQ  :=  TRUE;       //vent feeder
                   END_IF;

                   IF NOT ("DV".MOB_FDR_V24_OPN_REQ OR "PDO".V24) THEN
                       #step    :=  #step + 10;
                   END_IF;

               100://sequence aborted
                   //----------------
                   "LT".MOB_FDR_DCK_DONE :=  FALSE;
                   "LT".MOB_FDR_DCK_ATV  :=  FALSE;
                   "FLT".ME_LEAK_TST_FDR :=  FALSE;
                   #step                :=  0;

               110://finish sequence
                   //---------------
                   "LT".MOB_FDR_DCK_DONE :=  TRUE;
                   "LT".MOB_FDR_DCK_ATV  :=  FALSE;
                   "FLT".ME_LEAK_TST_FDR :=  FALSE;
                   #step                :=  0;

           END_CASE;

       ELSE
           #step    := 0;

       END_IF;
END_FUNCTION_BLOCK

FUNCTION_BLOCK "BM_MOB_FDR_UDCK"   // FB107, SCL
{ S7_Optimized_Access := 'FALSE' }
VERSION : 0.0
// --------------------------------------------------------------------------------
//     program     :   BM_MOB_FDR_UDCK
//     description :   undocking of mobile feeder from puller
//     name        :   G. Eibelsh鋟ser
//     date        :   26.10.2011
//   
//     revision    :
//     name        :
//     date        :    
//                     (c)PVATePla AG
//     --------------------------------------------------------------------------------
   VAR
      arb_udck_seq : Bool;
      fdr_prs_inc_done : Bool;
      "step" : Int;
      i : Int;
      prg_cnt : Int;
      fdr_prs_bfe_prs_drop : Real;
   END_VAR
   VAR CONSTANT
      up_prs_lim : Real := 90.0;
   END_VAR
BEGIN


       //set mobile feeder undocking request 
       //-----------------------------------
       IF      NOT "LT".MOB_FDR_DCK_ATV                                  //feeder docking sequence is not running
           AND NOT "LT".MOB_FDR_UDCK_DONE                                //undocking sequence is not done
           AND     "DV".FDR_TUBE_HOME_POS                             //feeder tube is in home position
           AND     "PDI".LS_V11_CL   THEN                                //valve V11 is closed

           IF "KYD".MOB_FDR_UDCK_ON THEN
               "LT".MOB_FDR_UDCK_ATV  :=  TRUE;
           END_IF;
       END_IF;

       //abort mobile feeder undocking sequence
       //--------------------------------------
       IF NOT "LT".MOB_FDR_UDCK_DONE AND NOT "FLT".MOB_FDR_UDCK_SEQ_ABR THEN
           IF "LT".MOB_FDR_UDCK_ATV AND "KYD".MOB_FDR_ARB_SEQ  THEN
               #arb_udck_seq  :=  true;
           END_IF;
       END_IF;

       //mobile feeder undocking sequence
       //--------------------------------
       IF "LT".MOB_FDR_UDCK_ATV  THEN 

           //set step to abort undocking sequence
           //------------------------------------
           IF #arb_udck_seq THEN
               #step    := 80;      //abort step
           END_IF;

           //sequence steps
           //--------------
           CASE #step OF 

               0 : //initialisation step
                   //-------------------
                   #i                           :=  0;
                   "AV".ACT_PRS_DROP_FDR         :=  0.0;
                   "FLT".ME_PRS_DROP_FDR         :=  FALSE;
                   "FLT".MOB_FDR_FNC_PRS_HI      :=  FALSE;
                   "FLT".MOB_FDR_PRS_HI          :=  FALSE;
                   "FLT".MOB_FDR_DCK_SEQ_ABR     :=  FALSE;
                   "FLT".MOB_FDR_UDCK_SEQ_ABR    :=  FALSE;
                   #fdr_prs_inc_done            :=  false;
                   #step                        :=  #step + 10;

               10: //check if feeder is already at atmospheric pressure
                   //--------------------------------------------------
                   IF "PDI".FDR_APS THEN
                       #step    :=  #step + 60;      //go to step 70 and finish sequence
                   ELSE
                       #step    :=  #step + 10;      //go to next step and check pressure
                   END_IF;

               20: //check if furnace and feeder pressure are in valid range for pressure drop test 
                   //------------------------------------------------------------------------------
                   (*
                   IF ((AV.ACT_PRS_CLF + CNF.MOB_FDR_PRS_INC) >= up_prs_lim) THEN
                       FLT.MOB_FDR_FNC_PRS_HI  :=  TRUE;   
                   ELSIF (AV.ACT_PRS_FDR >= up_prs_lim) THEN
                       FLT.MOB_FDR_PRS_HI  :=  TRUE;   
                   ELSE
                       step    :=  step + 10;      //go to next step and perform sequence
                   END_IF;
                   *)
                   //pressure range test skipped - pressure increase in step30 up to predefined value
                   //--------------------------------------------------------------------------------
                   #step    :=  #step + 10;      //go to next step and perform sequence

               30: //increase feeder pressure
                   //------------------------
                   IF (("AV".ACT_PRS_FDR >= "CNF".MOB_FDR_PRS_INC) OR #fdr_prs_inc_done) THEN
                       "DV".MOB_FDR_V24_OPN_REQ  :=  FALSE;      
                       #fdr_prs_inc_done        :=  true;
                       IF "SysTick1s"    THEN
                           #i := #i + 1;
                       END_IF;

                       IF (#i > 30) THEN                                    //wait 30 seconds
                           #fdr_prs_bfe_prs_drop    :=  "AV".ACT_PRS_FDR;     //store actual feeder pressure
                           #step                    :=  #step + 10;
                           #i                       :=  0;
                       END_IF;
                   ELSE
                       "DV".MOB_FDR_V24_OPN_REQ  :=  TRUE;       //insert gas
                   END_IF;

               40: //V11 pressure drop test
                   //----------------------
                   IF "SysTick1s"    THEN
                       #i := #i + 1;
                   END_IF;

                   //calculate feeder pressure drop
                   //------------------------------
                   "AV".ACT_PRS_DROP_FDR := #fdr_prs_bfe_prs_drop - "AV".ACT_PRS_FDR;

                   //pressure drop time over
                   //-----------------------
                   IF (#i >= (REAL_TO_INT("PAR_MAIN".MOB_FDR_UDCK_LKT_TME))) THEN
                       #step    :=  #step + 10;
                   END_IF;

               50: //set alarm message if pressure drop test failed
                   //----------------------------------------------
                   IF ("AV".ACT_PRS_DROP_FDR > "PAR_MAIN".MOB_FDR_UDCK_MAX_PRS_DRP) THEN
                       "FLT".ME_PRS_DROP_FDR :=  TRUE;       //pressure drop too large - leakage of valve V11

                       //repeat  pressure drop test
                       //----------------
                       IF "KYD".MOB_FDR_NEW_LKT   THEN
                           #step    :=  #step - 50;      //initialisation step 
                       END_IF;

                       //ignore bad leak rate
                       //--------------------
                       IF "KYD".MOB_FDR_IGN_LEAK_RTE   THEN
                           #step    :=  #step + 10;      //finish sequence
                       END_IF;

                       //abort sequence and vent feeder
                       //------------------------------
                       IF "KYD".MOB_FDR_ARB_SEQ   THEN
                           #step    :=  #step + 30;      //abort sequence
                       END_IF;

                   ELSE
                       #step    :=  #step + 10;              //finish sequence
                   END_IF;

               60: //vent feeder
                   //-----------
                   IF "DV".APS_FDR_DELAYED THEN                  //feeder at atmospheric pressure
                       "DV".MOB_FDR_V24_OPN_REQ  :=  FALSE;      //stop venting
                   ELSE 
                       "DV".MOB_FDR_V24_OPN_REQ  :=  TRUE;       //vent feeder
                   END_IF;

                   IF NOT ("DV".MOB_FDR_V24_OPN_REQ OR "PDO".V24)   THEN
                       #step    :=  #step + 10;
                   END_IF;

               70: //finish sequence
                   //---------------
                   "LT".MOB_FDR_UDCK_DONE    :=  TRUE;           //set set feeder undocking done flag
                   "LT".MOB_FDR_DCK_DONE     :=  FALSE;          //reset feeder docking done flag
                   "LT".MOB_FDR_UDCK_ATV     :=  FALSE;
                   "FLT".ME_PRS_DROP_FDR     :=  FALSE;
                   #step                    :=  0;

               80 ://sequence aborted
                   //----------------
                   "FLT".MOB_FDR_UDCK_SEQ_ABR    :=  TRUE;
                   "DV".MOB_FDR_V24_OPN_REQ      :=  FALSE;
                   "LT".MOB_FDR_UDCK_DONE        :=  FALSE;
                   "LT".MOB_FDR_UDCK_ATV         :=  FALSE;
                   #arb_udck_seq                :=  false;
                   #step                        :=  0;

           END_CASE;

       ELSE
           #step    := 0;

       END_IF;
END_FUNCTION_BLOCK

FUNCTION_BLOCK "BM_MOB_FDR_DRV_SEQ"   // FB108, SCL
{ S7_Optimized_Access := 'FALSE' }
VERSION : 0.0
// --------------------------------------------------------------------------------
//     program     :   BM_MOB_FDR_DRV_SEQ
//     description :   drive sequence of mobile feeder
//     name        :   G. Eibelsh鋟ser
//     date        :   31.10.2011
//   
//     revision    :
//     name        :
//     date        :    
//                     (c)PVATePla AG
//     --------------------------------------------------------------------------------
   VAR
      mob_fdr_mve_out_seq_on : Bool;
      fdr_prs_inc_done : Bool;
      i : Int;
      "step" : Int;
      mob_fdr_mve_out_dly : Int;
      cool_dn_stp : Int;
      act_tube_pos_bfe : Real;
   END_VAR
   VAR CONSTANT
      max_prs_hyst : Real := 5.0;   // [mbar]
      prs_inc : Real := 3.0;   // [mbar]
   END_VAR
BEGIN


       //activate feeder tube move sequences
       //-----------------------------------
       IF "LT".MOB_FDR_DCK_DONE THEN
           //trigger sequence abort
           //----------------------
           IF NOT "APC".AUTOMATIC AND ("LT".MOB_FDR_MVE_IN_SEQ_ON XOR "LT".MOB_FDR_MVE_OUT_SEQ_ON) THEN
               IF "KYD".MOB_FDR_MVE_SEQ_ARB OR NOT "PDI".EMO THEN 
                   "LT".MOB_FDR_MVE_SEQ_ARB  :=  TRUE;
               END_IF;
           END_IF;

           IF NOT ("LT".MOB_FDR_MVE_IN_SEQ_ON OR "LT".MOB_FDR_MVE_OUT_SEQ_ON) THEN     
               //automatic mode
               //--------------
               IF "APC".AUTOMATIC THEN
                   //trigger move in sequence
                   //------------------------
                   IF ("DC".MOB_FDR_MVE_IN_SEQ_ON AND NOT "DV".FDG_MVE_IN_SEQ_DONE) THEN
                       "LT".MOB_FDR_MVE_IN_SEQ_ON    :=  TRUE;
                       "LT".MOB_FDR_MVE_SEQ_ARB      :=  FALSE;
                       #step                        :=  0;
                   //trigger move out sequence
                   //------------------------
                   ELSIF ("DC".MOB_FDR_MVE_OUT_SEQ_ON AND NOT "DV".FDG_MVE_OUT_SEQ_DONE AND NOT "LT".MOB_FDR_VIB_ON) THEN
                       "LT".MOB_FDR_MVE_OUT_SEQ_ON   :=  TRUE;
                       "LT".MOB_FDR_MVE_SEQ_ARB      :=  FALSE;
                       #step                        :=  0;
                   END_IF;
               //manual mode
               //-----------
               ELSE
                   //trigger move in sequence
                   //------------------------
                   IF ("KYD".MOB_FDR_MVE_IN_SEQ_ON AND NOT "DV".FDG_MVE_IN_SEQ_DONE) THEN
                       "LT".MOB_FDR_MVE_IN_SEQ_ON    :=  TRUE;
                       "LT".MOB_FDR_MVE_SEQ_ARB      :=  FALSE;
                       #step                        :=  0;
                   //trigger move out sequence
                   //------------------------
                   ELSIF ("KYD".MOB_FDR_MVE_OUT_SEQ_ON AND NOT "DV".FDG_MVE_OUT_SEQ_DONE AND NOT "LT".MOB_FDR_VIB_ON) THEN
                       "LT".MOB_FDR_MVE_OUT_SEQ_ON   :=  TRUE;
                       "LT".MOB_FDR_MVE_SEQ_ARB      :=  FALSE;
                       #step                        :=  0;
                   END_IF;
               END_IF;
           END_IF;
       END_IF;

       //delay tube move out sequence start
       //----------------------------------
       #mob_fdr_mve_out_seq_on  := "SysOndelay"(  DIN     := "LT".MOB_FDR_MVE_OUT_SEQ_ON,   // trigger input
                                               SetTime := 30,                          // setp. time
                                               ActTime := #mob_fdr_mve_out_dly,         // act. time
                                               Tick    := "SysTick100ms");               // timebase (100ms)

       //quartz tube move in furnace sequence
       //------------------------------------
       IF "LT".MOB_FDR_MVE_IN_SEQ_ON THEN

           //abort move in sequence
           //----------------------
           IF "LT".MOB_FDR_MVE_SEQ_ARB THEN
               #step    :=  100;            //abort step
           END_IF;

           //sequence steps
           //-------------- 
           CASE #step OF 

               0 : //initialisation step
                   //-------------------
                   #i                           :=  0;
                   #step                        :=  #step + 10;
                   #fdr_prs_inc_done            :=  false;
                   "DV".FDG_MVE_OUT_SEQ_DONE     :=  FALSE;
                   "FLT".MOB_FDR_MOV_IN_SEQ_ABR  :=  FALSE;          //reset alarm message
                   "FLT".MOB_FDR_MOV_OUT_SEQ_ABR :=  FALSE;          //reset alarm message

               10: //check pressure
                   //--------------
                   IF (("AV".ACT_PRS_FDR <= ("AV".ACT_PRS_FCH + #max_prs_hyst)) OR "PDI".LS_V11_OP) THEN       //feeder pressure above puller pressure
                       #step    :=  #step + 30;      //switch to pressure equalisation step                   
                   ELSE
                       #step    :=  #step + 10;      //switch to next step                    
                   END_IF;

               20: //pump down feeder
                   //----------------
                   IF ("AV".ACT_PRS_FDR <= ("AV".ACT_PRS_FCH )) THEN   
                       "DV".MOB_FDR_V3_2_OPN_REQ :=  FALSE;                      //close valve V3.2
                       #step                    :=  #step + 10;                  //switch to next step
                   ELSE
                       "DV".MOB_FDR_P3_ON_REQ    :=  TRUE;                       //switch on pump
                       "DV".MOB_FDR_V3_2_OPN_REQ :=  TRUE;                       //open valve V3.2
                   END_IF;

               30: //wait 3sec.
                   //----------
                   IF NOT "PDO".V3_2 THEN                            //valve V3.2 closed
                       IF "SysTick1s" THEN
                           #i := #i + 1;                             //increase timer
                       END_IF;
                       IF (#i >= 3) THEN                            //wait 3 sec.
                           #step                    :=  #step + 10;  //switch to next step
                           "DV".MOB_FDR_P3_ON_REQ    :=  FALSE;      //switch off pump
                           #i                       :=  0;
                       END_IF;
                   END_IF;             

               40: //pressure equalisation feeder - puller
                   //-------------------------------------
                   IF (("AV".ACT_PRS_FDR >= ("AV".ACT_PRS_FCH + #prs_inc)) OR #fdr_prs_inc_done OR "PDI".LS_V11_OP)THEN  //feeder pressure above puller pressure
                       "DV".MOB_FDR_V24_OPN_REQ  :=  FALSE;      //request closing of V24
                       #fdr_prs_inc_done        :=  true;
                       IF NOT "PDO".V24 THEN                     //V24 closed
                           IF "SysTick1s" THEN
                               #i := #i + 1;                     //increase timer
                           END_IF;
                           IF (#i >= 3) THEN                    //wait 3 sec.
                               #step    :=  #step + 10;          //switch to next step
                               #i       :=  0;
                           END_IF;
                       END_IF;
                   ELSE
                       "DV".MOB_FDR_V24_OPN_REQ  :=  TRUE;       //request opening of V24
                   END_IF;

               50: //open valve V11
                   //--------------
                   "DV".MOB_FDR_V11_OPN_REQ  :=  TRUE;
                   "DV".MOB_FDR_V11_CLD_REQ  :=  FALSE;
                   IF "PDO".FDR_V11_OP THEN                          //V11 opened
                       IF "SysTick1s" THEN
                           #i := #i + 1;                         //increase timer
                       END_IF;
                       IF (#i >= 3) THEN                        //wait 3 sec.
                           #step    :=  #step + 10;              //switch to next step
                           #i       :=  0;
                       END_IF;
                   END_IF;

               60: //move quartz tube inside furnace
                   //-------------------------------
                   IF ("PDO".FDR_V11_OP AND "PDI".LS_V11_OP AND NOT "PDI".LS_V11_CL) THEN
                       IF "DV".FDR_TUBE_FCH_POS THEN
                           "DV".MVE_FDR_TUBE_DN  :=  FALSE;
                           IF "SysTick1s" THEN
                               #i := #i + 1;                     //increase timer
                           END_IF;
                           IF (#i >= 3) THEN                    //wait 3 sec.
                               #step    :=  #step + 10;          //switch to next step
                               #i       :=  0;
                           END_IF;
                       ELSE
                           "DV".MVE_FDR_TUBE_DN  :=  TRUE;
                       END_IF;
                   END_IF;         

               70: //move chute in feeding position
                   //-------------------------------
                   IF "DV".FDR_TUBE_FCH_POS THEN
                       IF "DV".FDR_CH_FDG_POS THEN
                           "DV".FDR_CH_SW_R  :=  FALSE;   
                           IF "SysTick1s" THEN
                               #i := #i + 1;                     //increase timer
                           END_IF;
                           IF (#i >= 3) THEN                    //wait 3 sec.
                               #step    :=  #step + 10;          //switch to next step
                               #i       :=  0;
                           END_IF;
                       ELSE
                           "DV".FDR_CH_SW_R  :=  TRUE;   
                       END_IF;
                   END_IF;

               80: //move quartz tube in feeding position
                   //------------------------------------
                   IF "DV".FDR_CH_FDG_POS THEN
                       IF "DV".FDR_TUBE_FDG_POS THEN
                           "DV".MVE_FDR_TUBE_UP  :=  FALSE;
                           IF "SysTick1s" THEN
                               #i := #i + 1;                     //increase timer
                           END_IF;
                           IF (#i >= 3) THEN                    //wait 3 sec.
                               #step    :=  #step + 10;          //switch to next step
                               #i       :=  0;
                           END_IF;
                       ELSE
                           "DV".MVE_FDR_TUBE_UP  :=  TRUE;
                       END_IF;
                   END_IF;         

              90:  //move in sequence done
                   //---------------------
                   "DV".FDG_MVE_IN_SEQ_DONE      :=  TRUE;       //set move in sequence done flag
                   "LT".MOB_FDR_MVE_IN_SEQ_ON    :=  FALSE;      //reset move in sequence on flag
                   #step                        :=  0;          //reset step number

              100: //abort move in sequence
                   //----------------------
                   "FLT".MOB_FDR_MOV_IN_SEQ_ABR  :=  TRUE;       //set alarm message
                   "LT".MOB_FDR_MVE_IN_SEQ_ON    :=  FALSE;      //reset move in sequence on flag
                   "DV".FDG_MVE_IN_SEQ_DONE      :=  FALSE;      //reset move in sequence done flag
                   "DV".MOB_FDR_V24_OPN_REQ      :=  FALSE;      //close valve V24 
                   "DV".MVE_FDR_TUBE_DN          :=  FALSE;      //stop tube drive down
                   "DV".MVE_FDR_TUBE_UP          :=  FALSE;      //stop tube drive up
                   "DV".FDR_CH_SW_R              :=  FALSE;      //stop chute drive swivel right
                   #step                        :=  0;          //reset step number

           END_CASE;

       END_IF;

       //quartz tube move out of furnace sequence
       //----------------------------------------
       IF #mob_fdr_mve_out_seq_on THEN
           //abort move out sequence
           //----------------------
           IF "LT".MOB_FDR_MVE_SEQ_ARB THEN
               #step    :=  80;            //abort step
           END_IF;

           //sequence steps
           //--------------    
           CASE #step OF 

               0 : //initialisation step
                   //-------------------
                   #i                           :=  0;
                   #cool_dn_stp                 :=  0;
                   #step                        :=  #step + 10;
                   "DV".FDG_MVE_IN_SEQ_DONE      :=  FALSE;
                   "FLT".MOB_FDR_MOV_OUT_SEQ_ABR :=  FALSE;       //reset alarm message
                   "FLT".MOB_FDR_MOV_IN_SEQ_ABR  :=  FALSE;       //reset alarm message

               10: //move quartz tube inside furnace (bypassed if chute is already in home position)
                   //-------------------------------------------------------------------------------
                   IF ("DV".FDR_TUBE_FCH_POS OR "DV".FDR_CH_HOME_POS) THEN
                       "DV".MVE_FDR_TUBE_DN  :=  FALSE;
                       IF "SysTick1s" THEN
                           #i := #i + 1;                         //increase timer
                       END_IF;
                       IF (#i >= 3) THEN                        //wait 3 sec.
                           #step    :=  #step + 10;              //switch to next step
                           #i       :=  0;
                       END_IF;
                   ELSE
                       "DV".MVE_FDR_TUBE_DN  :=  TRUE;
                   END_IF;

               20: //move chute in home position
                   //---------------------------
                   IF "DV".FDR_CH_HOME_POS THEN
                       "DV".FDR_CH_SW_L  :=  FALSE;   
                       IF "SysTick1s" THEN
                           #i := #i + 1;                         //increase timer
                       END_IF;
                       IF (#i >= 3) THEN                        //wait 3 sec.
                           #step    :=  #step + 10;              //switch to next step
                           #i       :=  0;
                       END_IF;
                   ELSE
                       "DV".FDR_CH_SW_L :=  TRUE;   
                   END_IF;

               30: //store tube position value
                   //-------------------------
                   #act_tube_pos_bfe    :=  "AV".MOB_FDR_ACT_TUBE_POS;  
                   #step                :=  #step + 10;                  //switch to next step
                   #i                   :=  0;
                   #cool_dn_stp         :=  #cool_dn_stp + 1;            //increase cool down step counter

               40: //move quartz tube in cool down steps upwards
                   //-------------------------------------------
                   IF (((REAL_TO_INT("PAR_MAIN".MOB_FDR_TUBE_COOL_STP) > 0) AND (REAL_TO_INT("PAR_MAIN".MOB_FDR_TUBE_TRV_INC) > 0))) THEN 
                       //switch tube upwards movement on/off
                       //-----------------------------------
                       IF (("AV".MOB_FDR_ACT_TUBE_POS <= (#act_tube_pos_bfe - "PAR_MAIN".MOB_FDR_TUBE_TRV_INC)) OR "DV".FDR_TUBE_HOME_POS) THEN
                           "DV".MVE_FDR_TUBE_UP  :=  FALSE;          //stop tube movement

                           IF "DV".FDR_TUBE_HOME_POS THEN
                               #step    :=  #step + 10;              //tube home position already reached - switch to next step
                           ELSE
                               IF "SysTick1s" THEN
                                   #i := #i + 1;                     //increase timer
                               END_IF;

                               //wait until cool down time is over
                               //---------------------------------
                               IF (#i >= REAL_TO_INT("PAR_MAIN".MOB_FDR_TUBE_COOL_DN_TME)) THEN                  
                                   //check if additional cool down step is requested
                                   //-----------------------------------------------
                                   IF (#cool_dn_stp >= (REAL_TO_INT("PAR_MAIN".MOB_FDR_TUBE_COOL_STP))) THEN  
                                       #step    :=  #step + 10;      //last cool down step done - move tube in home position
                                       #i       :=  0;
                                   ELSE
                                       #step    :=  #step - 10;      //additional cool down step follows        
                                       #i       :=  0;
                                   END_IF;
                               END_IF;
                           END_IF;  
                       ELSE
                           "DV".MVE_FDR_TUBE_UP  :=  TRUE;           //start tube movement
                       END_IF;
                       //check if Ar inlet during tube move out is requested
                       //---------------------------------------------------
                       "DV".MOB_FDR_V24_OPN_REQ  :=  (REAL_TO_INT("PAR_MAIN".MOB_FDR_COOL_V24_ON) = 1); 
                   ELSE
                       #step    :=  #step + 10;                      //move tube in home position
                   END_IF;

               50: //move quartz tube in home position
                   //---------------------------------
                   IF "DV".FDR_TUBE_HOME_POS THEN
                       "DV".MVE_FDR_TUBE_UP  :=  FALSE;
                       IF "SysTick1s" THEN
                           #i := #i + 1;                         //increase timer
                       END_IF;
                       IF (#i >= 3) THEN                        //wait 3 sec.
                           #step    :=  #step + 10;              //switch to next step
                           #i       :=  0;
                       END_IF;
                   ELSE
                       "DV".MVE_FDR_TUBE_UP      :=  TRUE;
                       //check if Ar inlet during tube move out is requested
                       //---------------------------------------------------
                       "DV".MOB_FDR_V24_OPN_REQ  :=  (REAL_TO_INT("PAR_MAIN".MOB_FDR_COOL_V24_ON) = 1); 
                   END_IF;

               60: //close valve V11
                   //---------------
                   "DV".MOB_FDR_V11_CLD_REQ  :=  TRUE;
                   "DV".MOB_FDR_V11_OPN_REQ  :=  FALSE;
                   IF (NOT "PDO".FDR_V11_OP AND "PDI".LS_V11_CL AND NOT "PDI".LS_V11_OP) THEN
                       "DV".MOB_FDR_V24_OPN_REQ  :=  FALSE;      //request closing of V24
                       IF "SysTick1s" THEN
                           #i := #i + 1;                         //increase timer
                       END_IF;
                       IF (#i >= 3) THEN                        //wait 3 sec.
                           #step    :=  #step + 10;              //switch to next step
                           #i       :=  0;
                       END_IF;
                   END_IF;

              70:  //move out sequence done
                   //----------------------
                   "DV".FDG_MVE_OUT_SEQ_DONE     :=  TRUE;       //set move out sequence done flag
                   "LT".MOB_FDR_MVE_OUT_SEQ_ON   :=  FALSE;      //reset move in sequence on flag
                   #step                        :=  0;          //reset step number

               80: //abort move out sequence
                   //----------------------
                   "FLT".MOB_FDR_MOV_OUT_SEQ_ABR :=  TRUE;       //set alarm message
                   "LT".MOB_FDR_MVE_OUT_SEQ_ON   :=  FALSE;      //reset move in sequence on flag
                   "DV".MOB_FDR_V24_OPN_REQ      :=  FALSE;      //close valve V24
                   "DV".FDG_MVE_OUT_SEQ_DONE     :=  FALSE;      //reset move in sequence done flag
                   "DV".MVE_FDR_TUBE_DN          :=  FALSE;      //stop tube drive down
                   "DV".MVE_FDR_TUBE_UP          :=  FALSE;      //stop tube drive up
                   "DV".FDR_CH_SW_L              :=  FALSE;      //stop chute drive swivel right
                   #step                        :=  0;          //reset step number

           END_CASE;
       END_IF;
END_FUNCTION_BLOCK

FUNCTION_BLOCK "BM_ACC_MAIN"   // FB111, SCL
{ S7_Optimized_Access := 'FALSE' }
VERSION : 0.0
// --------------------------------------------------------------------------------
//     program     :    BM_ACC_MAIN
//     description :    main function block of active crystal cooling      
//     name        :    G. Eibelsh鋟ser
//     date        :    07.08.2012
// 
//     revision    :
//     name        :
//     date        :    
//                     (c)PVA Tepla AG
//     --------------------------------------------------------------------------------
   VAR
      flash_light : Bool;
      sound : Bool;
      acc_ok : Bool;
      sc_reset : Bool;
      schall : Bool;
      fp_schall : Bool;
      edge_schall : Bool;
      ackn_sound : Bool;
      prs_check : Bool;
      prs_check_rst : Bool;
      key_on : Bool;
      wtr_flw_diff_mon : Bool;
      abort_ovp_test : Bool;
      aps_fch_dly_prv : Bool;
      acc_key_rst_prv : Bool;
      rst_ovp_test_dbl : Bool;
      acc_sc_wtr_ok_prv : Bool;
      sc_reset_dly : Int;
      wtr_flw_diff_mon_dly : Int;
      htr_off_tme : Int;
      ovp_test_tme : Int;
      ovp_rst_tme : Int;
      i : Int;
      j : Int;
      wtr_diff : Real;
      wtr_flw_in_sum : Real;
      wtr_flw_out_sum : Real;
      wtr_flw_in : Array[0..4] of Real;
      wtr_flw_out : Array[0..4] of Real;
   END_VAR
   VAR CONSTANT
      wtr_tmp_wrn : Real := 50.0;   // warning water outlet temperature of cooling coil [癈] - alarm message
      min_wtr_coil_prs : Real := 1.5;   // min. water cooling coil inlet pressure in [bar] - alarm message
      min_wtr_spl_prs : Real := 2.0;   // min. water supply inlet pressure in [bar] - alarm message
      min_wtr_flw : Real := 10.0;   // min. water flow in l/min - alarm message
      wtr_flw_diff_wrn : Real := 0.5;   // max. water flow deviation of inlet and outlet in [l/min] - alarm message
   END_VAR
BEGIN


       //display of cooling water temperature, pressure and flow - coming from analog inputs
       //-----------------------------------------------------------------------------------
       "DIS".ACC_WTR_TMP     := "PAI".ACC_WTR_TMP;                 //sensor: Kobold TMA PT100
       "DIS".ACC_WTR_PRS_IN  := "PAI".ACC_WTR_PRS_IN;              //sensor: B黵kert 8314
       "DIS".ACC_WTR_SPL_PRS := "PAI".ACC_WTR_SPL_PRS;             //sensor: B黵kert 8314
       "DIS".ACC_WTR_FLW_OUT := "PAI".ACC_WTR_FLW_OUT;             //sensor: Profimess SI00
       "DIS".ACC_WTR_FLW_IN  := "PAI".ACC_WTR_FLW_IN;              //sensor: Profimess SI00
     //DIS.ACC_WTR_DIFF    := PAI.ACC_WTR_FLW_IN - PAI.ACC_WTR_FLW_OUT;

       //calculation of flow difference after averaging of input variables
       //-----------------------------------------------------------------
       IF "SysTick100ms" THEN
           //store flow values
           //-----------------
           #wtr_flw_in[#i] := "PAI".ACC_WTR_FLW_IN;
           #wtr_flw_out[#i] := "PAI".ACC_WTR_FLW_OUT;
           //increase array counter
           //----------------------
           IF (#i < 4) THEN 
               #i   :=  #i + 1;
           //reset array counter
           //-------------------
           ELSE
               //reset counter and flow values
               //-----------------------------   
               #i := 0;
               #wtr_flw_in_sum  := 0.0; 
               #wtr_flw_out_sum := 0.0;
               //sum five values
               //---------------
               FOR #j := 0 TO 4 DO
                   #wtr_flw_in_sum  := #wtr_flw_in_sum + #wtr_flw_in[#j];
                   #wtr_flw_out_sum := #wtr_flw_out_sum + #wtr_flw_out[#j];
               END_FOR;
           END_IF;
       END_IF;

       //display flow difference
       //-----------------------    
       "DIS".ACC_WTR_DIFF    := (#wtr_flw_in_sum - #wtr_flw_out_sum) / 5;

       IF ("SY".RUN_TIME > 5) THEN               //PLC restarted
           //alarm message if water temperature reached the warning level - coming from analog input
           //---------------------------------------------------------------------------------------
           "FLT".ACC_WRN_WTR_TMP := ("PAI".ACC_WTR_TMP >= #wtr_tmp_wrn);       

           //alarm messages of water pressure and flow - coming from analog inputs
           //---------------------------------------------------------------------
           "FLT".ACC_WRN_WTR_PRS_IN  := ("PAI".ACC_WTR_PRS_IN  < #min_wtr_coil_prs);   
           "FLT".ACC_WRN_WTR_SPL_PRS := ("PAI".ACC_WTR_SPL_PRS < #min_wtr_spl_prs);    
           "FLT".ACC_WRN_WTR_FLW_OUT := ("PAI".ACC_WTR_FLW_OUT < #min_wtr_flw);        
           "FLT".ACC_WRN_WTR_FLW_IN  := ("PAI".ACC_WTR_FLW_IN  < #min_wtr_flw);     
           "FLT".ACC_WTR_DIFF        := (#wtr_flw_diff_mon AND ("DIS".ACC_WTR_DIFF >= #wtr_flw_diff_wrn));  

           //common alarms - coming from digital inputs
           //------------------------------------------
           "FLT".ACC_CB_FLT_DC24V        := NOT "PDI".ACC_CB_FLT_DC24V;
           "FLT".ACC_CB_FLT_AC230V       := NOT "PDI".ACC_CB_FLT_AC230V;
           "FLT".ACC_UPS_24V_ALM         := "PDI".ACC_UPS_24V_ALM;
           "FLT".ACC_UPS_BAT_MODE        := "PDI".ACC_UPS_24V_NRM;
           "FLT".ACC_WTR_PRS_COMP_TANK   := NOT "PDI".DPH_RPT_DET_OK;

           //St鰎ungen an 躡erdruckschaltern oder Trennverst鋜kern
           //-----------------------------------------------------
           "FLT".ACC_OVP_1_FLT := "PDI".OV_PRS_1_FLT;  
           "FLT".ACC_OVP_2_FLT := "PDI".OV_PRS_2_FLT;    

           //set alarm messages of serious faults
           //------------------------------------
           "FLT".ACC_WRN_FCH_OV_PRS_1    := NOT "PDI".ACC_FCH_OV_PRS_1;                    //over pressure switch 1    - Wika ?
           "FLT".ACC_WRN_FCH_OV_PRS_2    := NOT "PDI".ACC_FCH_OV_PRS_2;                    //over pressure switch 2    - Wika ?
           "FLT".ACC_WTR_FLW_IN          := NOT "PDI".ACC_WTR_FLW_IN_OK;                   //water inlet flow sensor   - sensor EGE SC10963
           "FLT".ACC_WTR_FLW_OUT         := NOT "PDI".ACC_WTR_FLW_OUT_OK;                  //water outlet flow sensor  - sensor EGE SC10963
           "FLT".ACC_WTR_TMP_OUT         := NOT "PDI".ACC_WTR_TMP_OUT_OK;                  //water temperature sensor  - Jumo Thermostat Typ ATHs 270

           //serious ACC faults - shut off of heater and water valves - coming from PNOZ
           //---------------------------------------------------------------------------
           "FLT".ACC_SC_WTR  := NOT "PDI".ACC_SC_WTR_OK;                                   // PNOZ +N9-13K2 ausgel鰏t
           "FLT".ACC_SC_HTR  := NOT "PDI".ACC_SC_HTR_OK;                                   // PNOZ +N9-14K4 ausgel鰏t

       END_IF;

       //enable water flow difference monitoring
       //---------------------------------------
       #wtr_flw_diff_mon    :=  "SysOndelay"( DIN     := "LT".ACC_SC_WTR_STR_ON,
                                           SetTime := 10,                      
                                           ActTime := #wtr_flw_diff_mon_dly,    // act. time
                                           Tick    := "SysTick1s");              // timebase (1s)  

       // activate pressure check
       //------------------------
       IF ("LT".HTR_1_ON AND "LT".P1_ON AND ("AV".ACT_PRS_FCH < 95.0)) THEN    
           #prs_check       := true;
       END_IF;    

       //monitor pressure increase
       //-------------------------
       IF (#prs_check AND "LT".V1_OPEN AND ("AV".ACT_PRS_FCH > 99.0)) THEN
           "FLT".ACC_EX_ALARM := TRUE;                           //set common alarm
       END_IF;

       //reset pressure increase alarm
       //-----------------------------
       IF ("DV".APS_FCH_DELAYED AND "DV".APS_GCH_DELAYED) THEN     //reset at atmospheric pressure
           "FLT".ACC_EX_ALARM := FALSE;
           #prs_check        := false;

       ELSIF ("AV".ACT_PRS_FCH < 99.0) THEN                      //reset below pressure limit
           "FLT".ACC_EX_ALARM := FALSE;
       END_IF;

       //delay flag pressure check reset 
       //-------------------------------
       #prs_check_rst := "SysOndelay"(DIN     := NOT "LT".HTR_1_ON,
                                   SetTime := 10800,               // delay 3h after heater off
                                   ActTime := #htr_off_tme,         // act. time
                                   Tick    := "SysTick1s");          // timebase (1s)

       //deactivate pressure monitoring
       //------------------------------
       IF (#prs_check_rst OR "DV".APS_FCH_DELAYED) THEN
           #prs_check := false;
       END_IF;

       //set alarm message when overpressure test was not done 
       //-----------------------------------------------------
       IF NOT "LT".SI_FIL_FSH_SEQ_ON THEN 
           IF NOT "DV".ACC_ENB_VAC AND (("KYA".SET_CTL_VALVE_POS >= 0.1) OR "KYD".STATE_RUN OR "KYD".MOD_AUTO) THEN  //open control valve or process start
               "FLT".MAKE_OVP_TEST := TRUE;    
           ELSE 
               "FLT".MAKE_OVP_TEST := FALSE;
           END_IF;
       ELSE 
           "FLT".MAKE_OVP_TEST := FALSE;
       END_IF;       

       //set alarm flag of light signal
       //------------------------------
       #flash_light   :=    "FLT".ACC_WRN_FCH_OV_PRS_1
                       OR  "FLT".ACC_WRN_FCH_OV_PRS_2 
                       OR  "FLT".ACC_WTR_TMP_OUT
                       OR  "FLT".ACC_WTR_FLW_IN 
                       OR  "FLT".ACC_WTR_FLW_OUT
                       OR  "FLT".ACC_EX_ALARM; 

       //set alarm flag of accustic signal
       //---------------------------------
       #schall  :=  "FLT".ACC_WRN_FCH_OV_PRS_1 AND "FLT".ACC_WRN_FCH_OV_PRS_2 OR
                   "FLT".ACC_WTR_FLW_IN AND "FLT".ACC_WTR_FLW_OUT AND NOT "DV".ACC_OVP_TEST_ON;                    

       //built positive edge impulse of alarm flag
       //-----------------------------------------
       #fp_schall   := #schall AND NOT #edge_schall;
       #edge_schall := #schall;

       //set sound on positive edge impulse
       //----------------------------------
       IF #fp_schall THEN
           #sound       := true;   
       END_IF;

       //reset sound
       //-----------
       IF #ackn_sound THEN
           #sound       := false;    
           #ackn_sound  :=  false;
       END_IF;

       IF "KYD".ALARM_ACKN AND #sound THEN
           #ackn_sound := true;    
       END_IF;

       // set alarm outputs
       //------------------
       "PDO".ACC_ALM_LT_1  :=  #flash_light;        
       "PDO".ACC_ALM_LT_2  :=  #flash_light;     
       "PDO".ACC_ALM_SND_1 :=  #sound;
       "PDO".ACC_ALM_SND_2 :=  #sound;   

       //enable ACC overpressure test - enables button on touch screen
       //-------------------------------------------------------------
       "LT".ACC_OVP_TEST_ENB :=      NOT "APC".AUTOMATIC  
                               AND     "DV".APS_GCH_DELAYED
                               AND     "DV".APS_FCH_DELAYED 
                               AND     "LT".V7_OPEN 
                              // AND    (PDI.LS_V11_CL OR NOT DV.MOB_FDR_V11_INST)   //feeder valve must be closed
                               AND     "PDI".LS_GCH_DN AND "PDI".LS_GCH_SW_IN          //gate chamber closed 
                               AND NOT "LT".V1_OPEN
                               AND NOT "LT".ACC_OVP_OK;

       //max. overpressure test time
       //---------------------------
       #abort_ovp_test  := "SysOndelay"(  DIN     := "DV".ACC_OVP_TEST_ON,
                                       SetTime := 30,                  // 30s
                                       ActTime := #ovp_test_tme,        // act. time
                                       Tick    := "SysTick1s");          // timebase (1s)

       //abort over pressure test - test failed
       //--------------------------------------
       IF (#abort_ovp_test OR NOT "PDI".EMO)  THEN               
           "DV".ACC_OVP_TEST_ON  := FALSE;       //stop overpressure test
           "FLT".ACC_OVP_TEST    := TRUE;        //set alarm overpressure test failed

       //stop overpressure test - test ok
       //--------------------------------
       ELSIF ("DV".ACC_OVP_TEST_ON AND NOT("PDI".ACC_FCH_OV_PRS_1 OR "PDI".ACC_FCH_OV_PRS_2)) THEN
           "DV".ACC_OVP_TEST_ON  := FALSE;     
           "LT".ACC_OVP_OK       := TRUE;        //set variable over pressure test ok  - enable button cooling water on
           "DV".ACC_ENB_VAC      := TRUE;        //enable vacuum process
           #rst_ovp_test_dbl    := true;        //reset of over pressure test is disabled

       //start overpressure test
       //-----------------------
       ELSIF "LT".ACC_OVP_TEST_ENB AND "KYD".ACC_OVP_TEST THEN
           "DV".ACC_OVP_TEST_ON  := TRUE;        
           "FLT".ACC_OVP_TEST    := FALSE;       //reset alarm overpressure test failed
       END_IF;

       //set light variable over pressure test on - reset delayed
       //--------------------------------------------------------
       "LT".ACC_OVP_TEST_ON  :=  "SysOffdelay"(DIN     := "DV".ACC_OVP_TEST_ON,
                                           SetTime := 10,                          // 1s
                                           ActTime := #ovp_rst_tme,                 // act. time
                                           Tick    := "SysTick100ms");               // timebase (100ms)

       //enable vacuum process after PLC restart
       //---------------------------------------
        IF ("SY".RUN_TIME < 5) THEN               //PLC restarted
           IF (NOT "PDI".FCH_APS AND ("AV".ACT_HTR_1_TMP >= ("CNF".HTR_1_TMP_RANGE_LOW + 20.0))) THEN    //furnace pressure low and heater hot
               "DV".ACC_ENB_VAC   := TRUE;  
           END_IF;
       END_IF;

       //reset variable over pressure test ok
       //------------------------------------
       IF ("DV".APS_FCH_DELAYED AND NOT #aps_fch_dly_prv) THEN            //normal reset when furnace is at atmospheric pressure 
           "LT".ACC_OVP_OK   := FALSE;  
           "DV".ACC_ENB_VAC  := FALSE;

       ELSIF (#acc_sc_wtr_ok_prv AND NOT "PDI".ACC_SC_WTR_OK AND NOT #rst_ovp_test_dbl) THEN  //reset after water flow fault in cooling coil
           "LT".ACC_OVP_OK   := FALSE;     
       END_IF;

       #aps_fch_dly_prv     :=  "DV".APS_FCH_DELAYED;     //store status of APS one cycle
       #acc_sc_wtr_ok_prv   :=  "PDI".ACC_SC_WTR_OK;      //store status of safety circuit water

       //enable switching of water and heater circuit with key switch
       //------------------------------------------------------------
       IF (("PDI".ACC_KEY_RST AND NOT #acc_key_rst_prv) AND NOT "LT".ACC_SC_WTR_STR_ON AND "LT".ACC_OVP_OK) THEN
           #key_on              := true;
           #rst_ovp_test_dbl    := false;       //reset of over pressure test is enabled

       END_IF;

       #acc_key_rst_prv :=  "PDI".ACC_KEY_RST;    //store status of key switch one cycle

       //enable ACC water start - enables button on touch screen
       //-------------------------------------------------------
       "LT".ACC_SC_WTR_STR_ENB   :=  #key_on;

       //activation of cooling water and heater circuit is enabled
       //---------------------------------------------------------
       IF #key_on THEN
           //close safety contacts cooling water and heater
           //----------------------------------------------                           
           IF "KYD".ACC_SC_WTR_STR THEN
               "PDO".ACC_SC_WTR_STR      := TRUE;            //set output safety circuit water start
               "PDO".ACC_SC_HTR_STR      := TRUE;            //set output safety circuit heater start
               "LT".ACC_SC_WTR_STR_ON    := TRUE;            //set light variable cooling water is on
           END_IF;   
       END_IF; 

       //delay setting of reset circuit
       //------------------------------
       #sc_reset := "SysOndelay"( DIN     := "PDI".ACC_SC_WTR_ATV AND "PDI".ACC_SC_HTR_ATV,
                               SetTime := 10,                          // setp. time
                               ActTime := #sc_reset_dly,                // act. time
                               Tick    := "SysTick100ms");               // timebase (100ms)     

       //reset safety circuit (PNOZ) of cooling water and heater
       //-------------------------------------------------------        
       IF #sc_reset THEN
           "PDO".ACC_SC_WTR_RST := TRUE;                    
           "PDO".ACC_SC_HTR_RST := TRUE;
       END_IF;

       IF "PDO".ACC_SC_WTR_RST THEN                      //safety circuit reset output active
           //reset water circuit output
           //--------------------------
           IF NOT "PDI".ACC_SC_WTR_ATV THEN              //momentary impulse of time based relais is over
               "PDO".ACC_SC_WTR_STR  := FALSE;
               "PDO".ACC_SC_WTR_RST  := FALSE;
           END_IF;
       END_IF;

       IF "PDO".ACC_SC_HTR_RST THEN                      //safety circuit reset output active
           //reset heater circuit output
           //---------------------------
           IF NOT "PDI".ACC_SC_HTR_ATV THEN              //momentary impulse of time based relais is over
               "PDO".ACC_SC_HTR_STR  := FALSE;
               "PDO".ACC_SC_HTR_RST  := FALSE;
           END_IF;
       END_IF;

       //reset light variable of water circuit
       //-------------------------------------  
       IF NOT "PDI".ACC_SC_WTR_OK AND NOT "PDO".ACC_SC_WTR_STR THEN     
           "LT".ACC_SC_WTR_STR_ON    := FALSE;                           //cooling water is off

       //reset key switch impulse
       //------------------------  
       ELSIF "PDI".ACC_SC_WTR_OK THEN     
           #key_on                  := false;                           //disable release of safety circuits from key swich
           "LT".ACC_SC_WTR_STR_ON    := TRUE;                            //cooling water is running
       END_IF;
END_FUNCTION_BLOCK

FUNCTION_BLOCK "BM_ACC_PRS_MON"   // FB112, SCL
{ S7_Optimized_Access := 'FALSE' }
VERSION : 0.0
// --------------------------------------------------------------------------------
//     program     :    BM_ACC_PRS_MON
//     description :    furnace pressure monitoring       
//     name        :    G. Eibelsh鋟ser
//     date        :    15.02.2013
// 
//     revision    :
//     name        :
//     date        :    
//                     (c)PVA Tepla AG
//     --------------------------------------------------------------------------------
   VAR
      enb_prs_mon : Bool;
      dbl_gas_valves : Bool;
      i : Int;
   END_VAR
   VAR CONSTANT
      opn_dly : Int := 60;   // delay reopening of gas inlet valves in sec.
      prs_hyst : Real := 50.0;   // pressure hysteries
   END_VAR
BEGIN

       //release gas inlet valves (V4, V5, V6) with time delay
       //-----------------------------------------------------    
       IF #dbl_gas_valves THEN
           //enable gas inlet valves (V4, V5, V6) after delay
           //------------------------------------------------
           IF (#i > #opn_dly) THEN
               "DV".ACC_ENB_GAS_V    :=  TRUE;
           //disable gas (V4, V5, V6) inlet valves
           //-------------------------------------
           ELSE
               "DV".ACC_ENB_GAS_V    :=  FALSE;
               //count 1s interval
               //-----------------
               IF "SysTick1s" THEN
                   #i := #i + 1;
               END_IF;
           END_IF;

       //release gas inlet valves (V4, V5, V6) immediadly
       //------------------------------------------------    
       ELSE
           "DV".ACC_ENB_GAS_V    :=  TRUE;
           #i                   :=  0;
       END_IF;

       //disable pressure monitoring
       //---------------------------
       IF ("DV".APS_GCH_DELAYED OR "LT".V7_CLOSE) THEN
           #enb_prs_mon    :=  false;
           #dbl_gas_valves :=  false;

       //enable pressure monitoring
       //--------------------------
       ELSIF ("AV".ACT_PRS_GCH < ("CNF".ACC_FNC_PRS_LIM - #prs_hyst)) THEN
           #enb_prs_mon    :=  true;
       END_IF;

